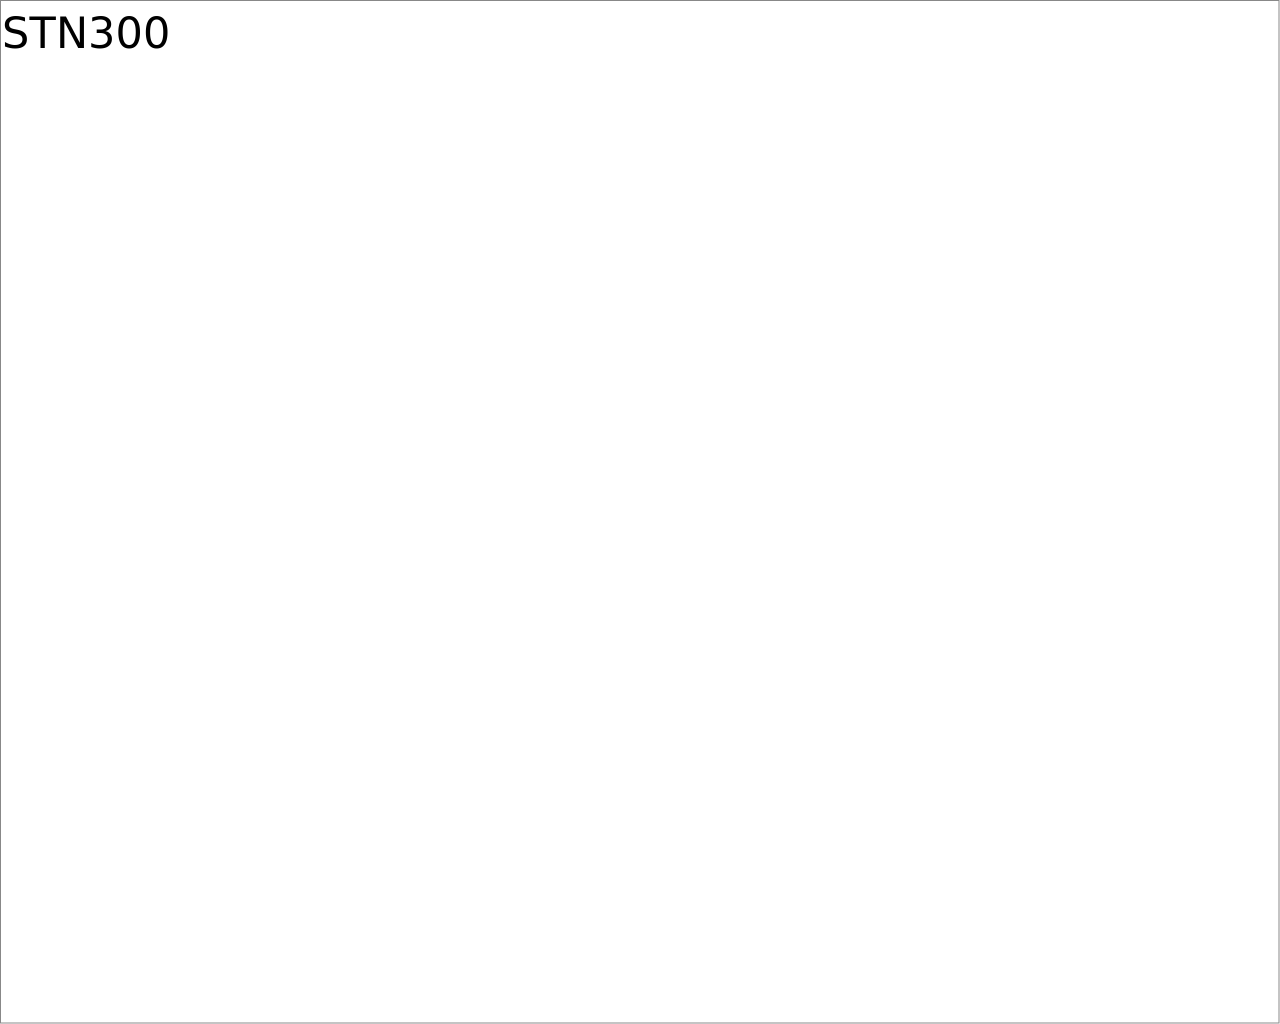
VISUALIZATION Visualization  // 1280x1024
    Label (1,3 171x60), "STN300"
END_VISUALIZATION

(* stored: Version 1.1.0.1, ProductVersion 3.1.4024.2
   Visu Visualization: Id {88f197ba-b36b-4758-886b-3858674ca2c2} *)
